FUNCTION_BLOCK FB_ReadGeophone
VAR_INPUT
	// none
END_VAR
VAR_OUTPUT
	velX : LREAL; // left -> right
	velY : LREAL; // back -> front
	velZ : LREAL; // top -> bottom
END_VAR
VAR
	c1Sample AT %I* : DINT; // channel 1 voltage (mV) -  x axis (yellow arrow)
	c2Sample AT %I* : DINT; // channel 2 voltage (mV) -  y axis (red arrow)
	c3Sample AT %I* : DINT; // channel 3 voltage (mV) -  z axis (rods -> level)
	
	// all real since need to be converted anyway
	peakVal : REAL := 10;
	maxInt : REAL := 7812500;
	sens : REAL := 78.9; // volts per meter per second
	unitMult : REAL := 1000; // m/s to mm/s
	mult : REAL := peakVal / maxInt / sens * unitMult;
END_VAR


// m/s
velX := DINT_TO_REAL(c1Sample) * mult;
velY := DINT_TO_REAL(c2Sample) * mult;
velZ := DINT_TO_REAL(c3Sample) * mult;

END_FUNCTION_BLOCK

(* stored: Version 1.1.0.1, ProductVersion 3.1.4024.13
   POU FB_ReadGeophone: Id {56b7d18b-71f0-4c3f-9840-fefa8f0a6997}, SpecialFunc None *)
